Yaskawa INFORM job: FRONT_WELD_90ST-2_5040.JBI

/JOB
//NAME FRONT_WELD_90ST-2_5040
///FOLDERNAME 02-SKRZYNIE_JOBS
//POS
///NPOS 17,17,0,4,0,0
///TOOL 0
///POSTYPE PULSE
///PULSE
C00000=0,-52278,40443,0,6873,1
C00001=0,-52278,40443,5610,-49281,-70968
C00002=0,-42686,23640,7425,-34877,-79161
C00003=-14116,-58141,-26117,-21696,-5351,-66126
C00004=-47175,-26068,-21336,-663,15689,-73543
C00005=-43679,-19644,-10767,-10092,13476,-68845
C00006=-35992,-25128,-16284,-12721,14581,-62558
C00007=-14522,-29408,-19323,-48383,21457,-43378
C00008=-14906,-39722,-32778,-45263,22245,-44952
C00009=-3902,-39042,-32149,-3317,17100,-71988
C00010=-3902,-39042,-32149,-3317,17100,-71988
C00011=-3867,-35433,-27527,-3373,17543,-71976
C00012=20137,-34393,-24870,-44565,22450,-50412
C00013=41669,-28424,-21699,-54677,35600,-43851
C00014=48063,-35826,-27915,-64657,37344,-38904
C00015=24039,-44019,6278,-32369,22109,-19464
C00016=0,-52278,40443,0,6873,1
BC00000=774759
BC00001=774759
BC00002=903040
BC00003=951614
BC00004=981280
BC00005=981280
BC00006=981280
BC00007=981280
BC00008=981280
BC00009=980954
BC00010=980954
BC00011=980954
BC00012=980954
BC00013=980954
BC00014=980954
BC00015=877951
BC00016=774759
///POSTYPE BASE
///RECTAN
///RCONF 0,0,0,0,0,0,0,0,0,0,0,0,0,0,0,0,0,0,0,0,0,0,0,0
P00501=-2.026,0.009,3.534,0.0000,0.0000,0.0000
///RCONF 1,0,0,0,0,0,0,0,0,0,0,0,0,0,0,0,0,0,0,0,0,0,0,0
P00502=-2.023,0.001,1.732,0.0000,0.0000,0.0000
P00503=0.138,-0.044,1.539,0.0000,0.0000,0.0000
P00504=-0.309,-0.010,1.636,0.0000,0.0000,0.0000
//INST
///DATE 2024/05/15 12:20
///ATTR SC,RW
///GROUP1 RB1,BS1
NOP
MOVJ C00000 BC00000 VJ=50.00
MOVJ C00001 BC00001 VJ=50.00
MOVJ C00002 BC00002 VJ=50.00
MOVJ C00003 BC00003 VJ=50.00
'::::::::::::::::::::::::::::::::
'W56
'::::::::::::::::::::::::::::::::
MOVL C00004 BC00004 V=666.7
SFTON P0501
MACRO1 MJ#(0) ARGF14
MOVL C00005 BC00005 V=166.7 PL=0
ARCON
MOVL C00006 BC00006 V=9.5
SFTOF
SFTON P0502
MOVL C00007 BC00007 V=9.5
ARCOF
MOVL C00008 BC00008 V=333.3
SFTOF
MOVL C00009 BC00009 V=333.3
'::::::::::::::::::::::::::::::::
'W21
'::::::::::::::::::::::::::::::::
MOVL C00010 BC00010 V=166.7
SFTON P0503
MACRO1 MJ#(0) ARGF14
MOVL C00011 BC00011 V=166.7 PL=0
ARCON
MOVL C00012 BC00012 V=9.5
SFTOF
SFTON P0504
MOVL C00013 BC00013 V=9.5
ARCOF
MOVL C00014 BC00014 V=250.0
SFTOF
MOVJ C00015 BC00015 VJ=50.00
MOVJ C00016 BC00016 VJ=50.00
END
